# EPICS substitutions: tpmacApp/pmc/xf10ida-mc02-brake.substitutions
file "PLC_brake.pmc"
{
pattern
{ PLC,  BRAKE,  MOTOR,  APPLY,  RELEASE }
{ 16,   32,     1,      0,      1  }
}
